
FUNCTION CB_bool_to_byte : BYTE


TITLE = ' Convert a boolean into an BYTE '
VERSION : '1.0'
AUTHOR  : CB
NAME    : boToByte
FAMILY  : TNI

VAR_INPUT
    IN : BOOL;
END_VAR

VAR_TEMP

END_VAR

BEGIN

CB_bool_to_byte := BOOL_TO_BYTE(IN);

END_FUNCTION
